// TwinCAT 3 PLC project AxisProgramming
// ProgramVersion: 3.1.4023.0
// libraries:
//   Tc2_MC2, * (Beckhoff Automation GmbH)
//   Tc2_NC, * (Beckhoff Automation GmbH)
//   Tc2_NCI, * (Beckhoff Automation GmbH)
//   Tc2_PlcInterpolation, * (Beckhoff Automation GmbH)
//   Tc2_Standard, * (Beckhoff Automation GmbH)
//   Tc2_System, * (Beckhoff Automation GmbH)
//   Tc3_Module, * (Beckhoff Automation GmbH)
// project tree:
//   DigitalSensor/ Digital_Input.TcPOU
//   DUTs/ AxisFBStatus.TcDUT, MC_Halt_Status.TcDUT, MC_Power_Status.TcDUT
//   GVLs/ AXIS_Declaration.TcGVL, Digital_Inputs.TcGVL
//   MasterAxis/ Master_Axis.TcPOU
//   / PlcTask.TcTTO
//   POUs/ MAIN.TcPOU
// real-time tasks:
//   TASK PlcTask: cycle T#10ms, priority 20, ADS port 350
// motion (NC):
//   TASK NC-Task 1 SAF: cycle T#2ms, priority 4, ADS port 501
//   TASK NC-Task 1 SVB: cycle T#10ms, priority 8, ADS port 511
//   AXIS Axis 1 (id 1)
//     OtherSettings: AllowMotionCmdToSlave=true
//     encoder EncType=1
//     drive DrvType=5
//       Analog: TorqueSetpointScale=10, ScaleFactorActTorque=0.1
//       TimeComp: TaskDelayCycles=1
//     controller CtrType=1
//       CtrPara: PriorControlFactor=1
//         Observer: BandWidth=20
//   AXIS Axis 2 (id 2)
//     OtherSettings: AllowMotionCmdToSlave=true
//     encoder EncType=1
//     drive DrvType=5
//       Analog: TorqueSetpointScale=10, ScaleFactorActTorque=0.1
//       TimeComp: TaskDelayCycles=1
//     controller CtrType=1
//       CtrPara: PriorControlFactor=1
//         Observer: BandWidth=20
//   AXIS Axis 3 (id 3)
//     OtherSettings: AllowMotionCmdToSlave=true
//     encoder EncType=1
//     drive DrvType=5
//       Analog: TorqueSetpointScale=10, ScaleFactorActTorque=0.1
//       TimeComp: TaskDelayCycles=1
//     controller CtrType=1
//       CtrPara: PriorControlFactor=1
//         Observer: BandWidth=20
// variable links:
//   AxisProgramming/AxisProgramming Instance <-> NC-Task 1 SAF/Axes/Axis 1
//     PlcTask Inputs/MAIN.AXIS_X.Linked_Axis.NcToPlc <-> Outputs/ToPlc
//     PlcTask Outputs/MAIN.AXIS_X.Linked_Axis.PlcToNc <-> Inputs/FromPlc
//   AxisProgramming/AxisProgramming Instance <-> NC-Task 1 SAF/Axes/Axis 2
//     PlcTask Inputs/AXIS_Declaration.Axis_Y.NcToPlc <-> Outputs/ToPlc
//     PlcTask Outputs/AXIS_Declaration.Axis_Y.PlcToNc <-> Inputs/FromPlc
//   AxisProgramming/AxisProgramming Instance <-> NC-Task 1 SAF/Axes/Axis 3
//     PlcTask Inputs/AXIS_Declaration.Axis_Z.NcToPlc <-> Outputs/ToPlc
//     PlcTask Outputs/AXIS_Declaration.Axis_Z.PlcToNc <-> Inputs/FromPlc

CONFIGURATION AxisProgramming
    RESOURCE PLC ON TwinCAT3
        TASK PlcTask(INTERVAL := T#10ms, PRIORITY := 20);
        PROGRAM MAIN WITH PlcTask : MAIN;
    END_RESOURCE
END_CONFIGURATION

// ---- DUTs/AxisFBStatus.TcDUT
TYPE AxisFBStatus :
STRUCT
	Power			: MC_Power_Status;
	Hault			: MC_Halt_Status;
END_STRUCT
END_TYPE

// ---- DUTs/MC_Halt_Status.TcDUT
TYPE MC_Halt_Status :
STRUCT
	Done           : BOOL;
    Busy           : BOOL;
    Active         : BOOL;
    CommandAborted : BOOL;
    Error          : BOOL;
    ErrorID        : UDINT;
END_STRUCT
END_TYPE

// ---- DUTs/MC_Power_Status.TcDUT
TYPE MC_Power_Status :
STRUCT
	Status		: BOOL;
	Busy		: BOOL;
	Active		: BOOL;
	Error		: BOOL;
	ErrorID		: UDINT;
END_STRUCT
END_TYPE

// ---- GVLs/AXIS_Declaration.TcGVL
{attribute 'qualified_only'}
VAR_GLOBAL
//	Axis_X		: AXIS_REF;
//	Axis_Y		: AXIS_REF;
//	Axis_Z		: AXIS_REF;
END_VAR

// ---- GVLs/Digital_Inputs.TcGVL
{attribute 'qualified_only'}
VAR_GLOBAL
	Axis1_Sensor1			: BOOL;
	Axis1_Sensor2			: BOOL;
	Axis2_Sensor1			: BOOL;
	Axis2_Sensor2			: BOOL;
	Axis3_Sensor1			: BOOL;
	Axis3_Sensor2			: BOOL;
END_VAR

// ---- POUs/MAIN.TcPOU
PROGRAM MAIN
VAR
	// Variables to call the axis
	AXIS_X		: Master_Axis;
	Axis_is_enabled	: BOOL;
	
	//Variables for axis Home
	Ref	: BOOL;
	Axis_is_at_Home : BOOL;
	
	//Variables of move absolute functions
	MoveAbsoluteDone : BOOL;
	StartMoveAbsolute : BOOL;
	
	//Variables of move relative functions
	MoveRelativeDone : BOOL;
	StartMoveRelative : BOOL;
	
	//Pause the axis while it is moving
	Pause_the_Axis	: BOOL;
	Pause_is_Done	: BOOL;
	
	
END_VAR

AXIS_X ();

AXIS_X.Enable();

IF AXIS_X.Enable() THEN
	Axis_is_enabled := TRUE;
END_IF


//Logic for referencing
IF Ref THEN
 	AXIS_X.Home();

	IF AXIS_X.Home() THEN
	Axis_is_at_Home := TRUE;	
	END_IF
	
END_IF

//Logic for move absolute
IF StartMoveAbsolute THEN
	AXIS_X.MoveAbsolute();
	
	IF AXIS_X.MoveAbsolute() THEN
		MoveAbsoluteDone := TRUE;
		StartMoveAbsolute := FALSE;
	END_IF
END_IF

// Logic for move relative
IF StartMoveRelative THEN
	AXIS_X.MoveRelative();
	
	IF AXIS_X.MoveRelative() THEN
		MoveRelativeDone := TRUE;
		StartMoveRelative := FALSE;
	END_IF
END_IF

// Pause the axis while moving

IF Pause_the_Axis THEN
	AXIS_X.Hault();
	
	IF AXIS_X.Hault() THEN
		Pause_is_Done := TRUE;
	END_IF
END_IF

END_PROGRAM

// ---- MasterAxis/Master_Axis.TcPOU
FUNCTION_BLOCK Master_Axis
VAR_INPUT
	Linked_Axis		: REF_AXIS;
END_VAR
VAR_OUTPUT
END_VAR
VAR
	// Motion Control Function Blocks
	Enable			: MC_POWER;
	Hault			: MC_HALT;
	Home			: MC_HOME;
	MoveAbsolute	: MC_MOVEABSOLUTE;
	MoveRelative	: MC_MOVERELATIVE;
	Stop			: MC_STOP;
	
	// Variables to operate functions of the axis
	PowerUp			: BOOL;
	Enable_Positive	: BOOL;
	Enable_Negative : BOOL;
	PowerOverride	: INT;
	PowerDown		: BOOL;
	
	Hault_Execute	: BOOL;
	HaultTrigger	: R_Trig;
	
	
	//Structure that hold variables which are connected wirh the output side of the MC FBs
	Status 			: AxisFBStatus;
	
	// State Machine Variable for axis
	State			:	INT;
END_VAR
VAR CONSTANT

END_VAR

Enable(Axis := Linked_Axis,
	   Enable:= Powerup,
	   Enable_Positive := Enable_Positive,
	   Enable_Negative := Enable_Negative,
	   Override := PowerOverride ,
	   BufferMode := ,
	   Options := ,
	   Status => Status.Power.Status,
	   Busy => Status.Power.Busy,
	   Active => Status.Power.Active,
	   Error => Status.Power.Error,
	   ErrorID => Status.Power.ErrorID);
	   
HaultTrigger(CLK := Hault_Execute);
	   
Hault(Execute := HaultTrigger.Q,
	  Deceleration := ,
	  Jerk := ,
	  BufferMode := ,
	  Options := ,
	  Done => Status.Hault.Done ,
	  Busy => Status.Hault.Busy ,
	  Active => Status.Hault.Active,
	  CommandAborted => Status.Hault.CommandAborted,
	  Error => Status.Hault.Error,
	  ErrorID => Status.Hault.ErrorID);

PROPERTY Axis_State : BOOL
GET
END_GET
SET
END_SET
END_PROPERTY

METHOD Enable
VAR_INPUT
END_VAR
END_METHOD

METHOD Hault
VAR_INPUT
END_VAR
END_METHOD

METHOD Home
VAR_INPUT
END_VAR
END_METHOD

METHOD MoveAbsolute 
VAR_INPUT
END_VAR
END_METHOD

METHOD MoveRelative : BOOL
VAR_INPUT
END_VAR
END_METHOD

METHOD Stop
VAR_INPUT
END_VAR
END_METHOD

END_FUNCTION_BLOCK

// ---- DigitalSensor/Digital_Input.TcPOU
FUNCTION_BLOCK Digital_Input
VAR_INPUT
	Input		: BOOL;
END_VAR
VAR_OUTPUT
END_VAR
VAR
END_VAR

PROPERTY PUBLIC Status : BOOL
GET
Status := Input;
END_GET
END_PROPERTY

END_FUNCTION_BLOCK
